// TIA Portal project "AWL LIBRO 4" (V11)

(* hardware
DEVICE "S7300/ET200 station_1"  SIMATIC 300-Station
   slot 0: "Perfil soporte_0"  Rail  6ES7 390-1***0-0AA0
   slot 2: "PLC_1"  CPU 313C-2 DP  6ES7 313-6CF03-0AB0  V2.6
      slot 0: "Interfaz MPI_1"  MPI
      slot 1: "Interfaz DP_1"  DP
      slot 2: "DI16/DO16_1"  DI16/DO16
      slot 4: "Contaje_1"  Counter
*)

// ===== PLC "PLC_1"  CPU 313C-2 DP =====

VAR_GLOBAL   // PLC tag table "Tabla de variables estándar"
   "FC S2 ABAJO" AT %E0.0 : Bool;
   "FC S3 ARRIBA" AT %E0.1 : Bool;
   "FC S4 IZQUIERDA" AT %E0.2 : Bool;
   "FC S5 DERECHA" AT %E0.3 : Bool;
   "MOTOR 1 SUBIR" AT %A0.0 : Bool;
   "MOTOR 1 BAJAR" AT %A0.1 : Bool;
   "MOTOR 2 DERECHA" AT %A0.2 : Bool;
   "MOTOR 2 IZQUIERDA" AT %A0.3 : Bool;
   "MARCHA" AT %E0.4 : Bool;
   "Tag_1" AT %M10.0 : Bool;
   "SALIDAS" AT %AB0 : Byte;
   "Tag_2" AT %M0.0 : Bool;
   "Tag_3" AT %T0 : Timer;
   "CONTROL" AT %MB1 : Byte;
   "Tag_4" AT %M1.0 : Bool;
   "Tag_5" AT %M1.1 : Bool;
   "Tag_6" AT %M1.2 : Bool;
   "Tag_7" AT %M1.3 : Bool;
   "Tag_8" AT %M1.7 : Bool;
   "Tag_9" AT %M0.1 : Bool;
END_VAR

ORGANIZATION_BLOCK "Main"   // OB1, STL
TITLE = EJERCICIO LIBRO 4. / "Main Program Sweep (Cycle)"
{ S7_Optimized_Access := 'FALSE' }
VERSION : 0.1
   VAR_TEMP
      OB1_EV_CLASS : Byte;   // Bits 0-3 = 1 (Coming event), Bits 4-7 = 1 (Event class 1)
      OB1_SCAN_1 : Byte;   // 1 (Cold restart scan 1 of OB 1), 3 (Scan 2-n of OB 1)
      OB1_PRIORITY : Byte;   // Priority of OB Execution
      OB1_OB_NUMBR : Byte;   // 1 (Organization block 1, OB1)
      OB1_RESERVED_1 : Byte;   // Reserved for system
      OB1_RESERVED_2 : Byte;   // Reserved for system
      OB1_PREV_CYCLE : Int;   // Cycle time of previous OB1 scan (milliseconds)
      OB1_MIN_CYCLE : Int;   // Minimum cycle time of OB1 (milliseconds)
      OB1_MAX_CYCLE : Int;   // Maximum cycle time of OB1 (milliseconds)
      OB1_DATE_TIME : Date_And_Time;   // Date and time OB1 started
   END_VAR
BEGIN

REGION Network 1
         A     "MARCHA";  // CUANDO ESTEN PRESIONADOS LOS FC PUEDES INICIAR CICLO 1.
         A     "FC S2 ABAJO";
         A     "FC S4 IZQUIERDA";
         FP    "Tag_1";
         JNB   _001;
         L     B#16#1;  // SUBIDA DE GRUA.
         T     "CONTROL";
   _001: NOP   0;
         A     "FC S4 IZQUIERDA";  // CUANDO ESTEN PRESIONADOS INICIARA EL DESPLAZMIENTO A LA DERECHA.
         A     "FC S3 ARRIBA";
         A     "MOTOR 1 SUBIR";
         JNB   _002;
         L     B#16#04;  // DESPLAZAMIENTO DE GRUA HACIA LA DERECHA.
         T     "CONTROL";
   _002: NOP   0;
         A     "FC S3 ARRIBA";  // CUANDO ESTEN PRESIONADOS INICIARA LA BAJADA.
         A     "FC S5 DERECHA";
         A     "MOTOR 2 DERECHA";
         JNB   _003;
         L     B#16#02;  // BAJADA GRUA.
         T     "CONTROL";
   _003: NOP   0;
         A     "FC S5 DERECHA";  // CUANDO ESTEN PRESIONADOS PARA LA GRUA Y TEMPORIZA CAMBIO A CICLO 2.
         A     "FC S2 ABAJO";
         =     "Tag_2";  // BOBINA ALIMENTACION T0.
         JNB   _004;
         L     B#16#00;  // PARO DE GRUA.
         T     "CONTROL";
   _004: NOP   0;
         A     "Tag_2";  // CONTACTO ALIMENTACION T0.
         L     S5T#4S;  // TEMPORIZADO 4S.
         SD    "Tag_3";  // T0.
         A     "Tag_3";  // CONTACTO TEMPORIZADO.
         JNB   _005;
         L     B#16#1;  // INICIO CICLO 2 SUBIDA GRUA.
         T     "CONTROL";
   _005: NOP   0;
         R     "Tag_2";
         S     "Tag_9";
         A     "FC S3 ARRIBA";  // CUANDO ESTEN PRESIONADOS INICIARA EL DESPLAZAMIENTO HACIA LA IZQUIERDA.
         A     "FC S5 DERECHA";
         A     "MOTOR 1 SUBIR";
         JNB   _006;
         L     B#16#08;  // DESPLAZAMIENTO DE GRUA HACIA LA IZQUIERDA.
         T     "CONTROL";
   _006: NOP   0;
         A     "FC S3 ARRIBA";  // CUANDO ESTEN PRESIONADOS INICIARA LA BAJADA.
         A     "FC S4 IZQUIERDA";
         A     "MOTOR 2 IZQUIERDA";
         JNB   _007;
         L     B#16#02;  // BAJADA GRUA
         T     "CONTROL";
   _007: NOP   0;
         A     "FC S2 ABAJO";
         A     "FC S4 IZQUIERDA";
         A     "MOTOR 1 BAJAR";
         JNB   _008;
         L     B#16#00;  // FIN DE CICLO SE PARA PARA VOLVER A ARRANCAR CUANDO SE PRECISE.
         T     "CONTROL";
   _008: NOP   0;



         A     "Tag_4";
         =     "MOTOR 1 SUBIR";
         A     "Tag_5";
         =     "MOTOR 1 BAJAR";
         A     "Tag_6";
         =     "MOTOR 2 DERECHA";
         A     "Tag_7";
         =     "MOTOR 2 IZQUIERDA";
END_REGION
END_ORGANIZATION_BLOCK